// LS Electric XG5000 project: fafasdf
// PLC LSPLC
// module base 0 slot 0: 입출력 모듈:XBC-DR32H (DC 24V 입력, 릴레이 출력 32점)
// module base 0 slot 1: 위치결정 모듈:XBF-PD02A (위치결정 펄스(LD)출력형, 2축)
// module base 0 slot 2: 출력 모듈:XBE-TN/TP16A (트랜지스터 출력, 16점 (싱크출력/소스출력))

PROGRAM NewProgram (task: 스캔 프로그램)

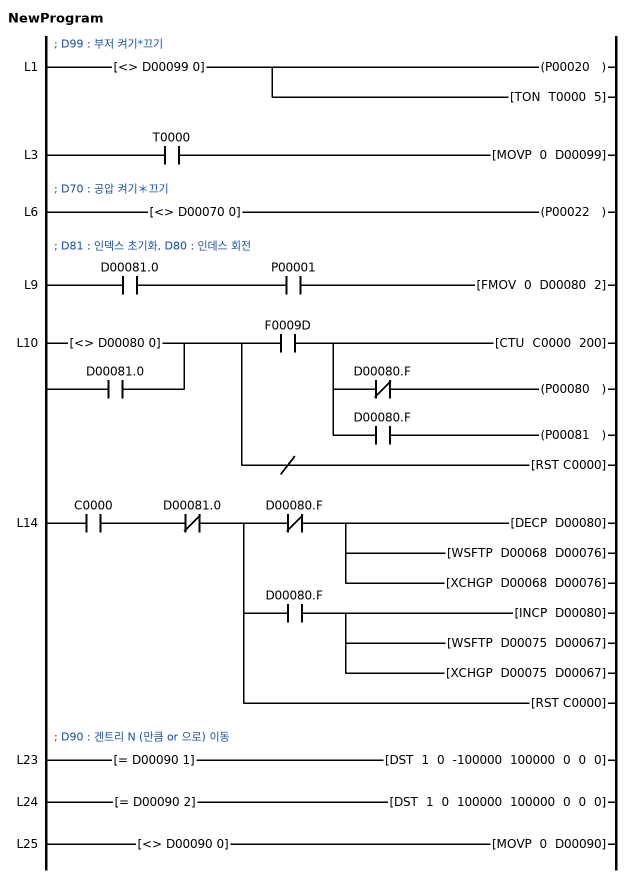
// D99 : 부저 켜기*끄기
; L1
LOAD<>    D00099 0
OUT       P00020
TON       T0000 5
; L3
LOAD      T0000
MOVP      0 D00099
// D70 : 공압 켜기＊끄기
; L6
LOAD<>    D00070 0
OUT       P00022
// D81 : 인덱스 초기화, D80 : 인데스 회전
; L9
LOAD      D00081.0
AND       P00001
FMOV      0 D00080 2
; L10
LOAD<>    D00080 0
OR        D00081.0
MPUSH
AND       F0009D
CTU       C0000 200
MPUSH
AND NOT   D00080.F
OUT       P00080
MPOP
AND       D00080.F
OUT       P00081
MPOP
NOT
RST       C0000
; L14
LOAD      C0000
AND NOT   D00081.0
MPUSH
AND NOT   D00080.F
DECP      D00080
WSFTP     D00068 D00076
XCHGP     D00068 D00076
MLOAD
AND       D00080.F
INCP      D00080
WSFTP     D00075 D00067
XCHGP     D00075 D00067
MPOP
RST       C0000
// D90 : 겐트리 N (만큼 or 으로) 이동 
; L23
LOAD=     D00090 1
DST       1 0 -100000 100000 0 0 0
; L24
LOAD=     D00090 2
DST       1 0 100000 100000 0 0 0
; L25
LOAD<>    D00090 0
MOVP      0 D00090